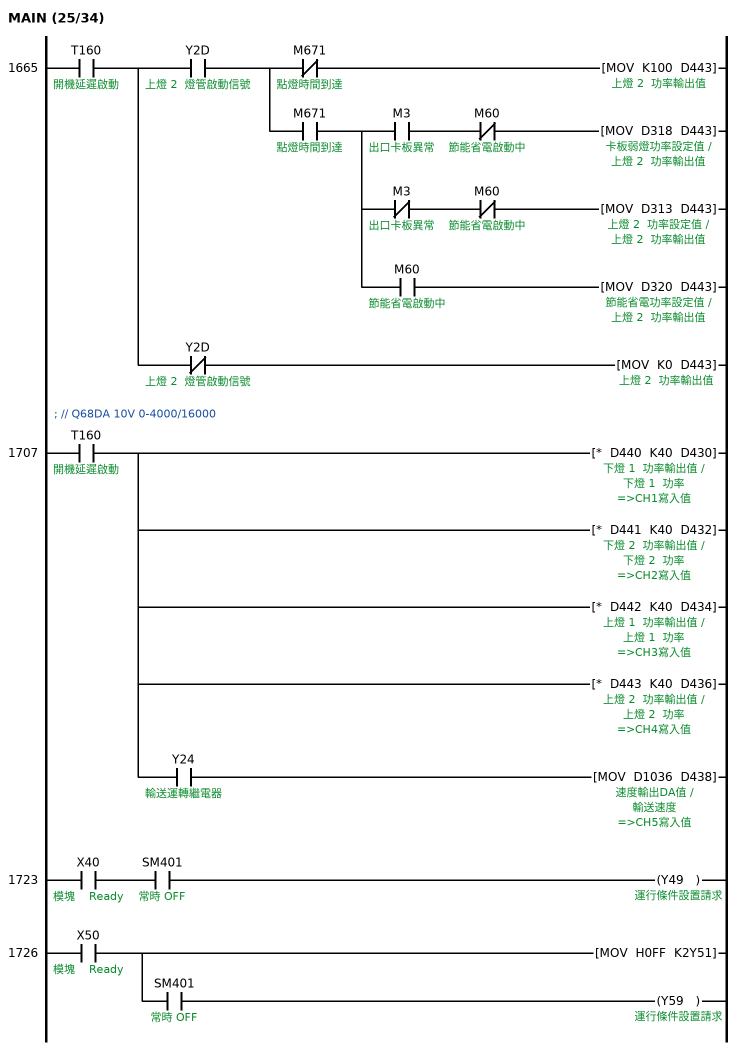
[picture p24: ladder of MAIN, rungs at steps 1665 to 1726]
1665  LD      T160  ; 開機延遲啟動
      MPS
      AND     Y2D  ; 上燈 2  燈管啟動信號
      MPS
      ANI     M671  ; 點燈時間到達
      MOV     K100 D443  ; 上燈 2  功率輸出值
      MPP
      AND     M671  ; 點燈時間到達
      MPS
      AND     M3  ; 出口卡板異常
      ANI     M60  ; 節能省電啟動中
      MOV     D318 D443
      MRD
      ANI     M3  ; 出口卡板異常
      ANI     M60  ; 節能省電啟動中
      MOV     D313 D443
      MPP
      AND     M60  ; 節能省電啟動中
      MOV     D320 D443
      MPP
      ANI     Y2D  ; 上燈 2  燈管啟動信號
      MOV     K0 D443
; // Q68DA 10V 0-4000/16000
1707  LD      T160  ; 開機延遲啟動
      *       D440 K40 D430  ; 下燈 1  功率  =>CH1寫入值
      *       D441 K40 D432  ; 下燈 2  功率  =>CH2寫入值
      *       D442 K40 D434  ; 上燈 1  功率  =>CH3寫入值
      *       D443 K40 D436  ; 上燈 2  功率  =>CH4寫入值
      AND     Y24  ; 輸送運轉繼電器
      MOV     D1036 D438  ; 速度輸出DA值 / 輸送速度      =>CH5寫入值
1723  LD      X40  ; 模塊    Ready
      AND     SM401  ; 常時 OFF
      OUT     Y49  ; 運行條件設置請求
1726  LD      X50  ; 模塊    Ready
      MOV     H0FF K2Y51  ; CH1輸出 允許/禁止標誌
      AND     SM401  ; 常時 OFF
      OUT     Y59  ; 運行條件設置請求
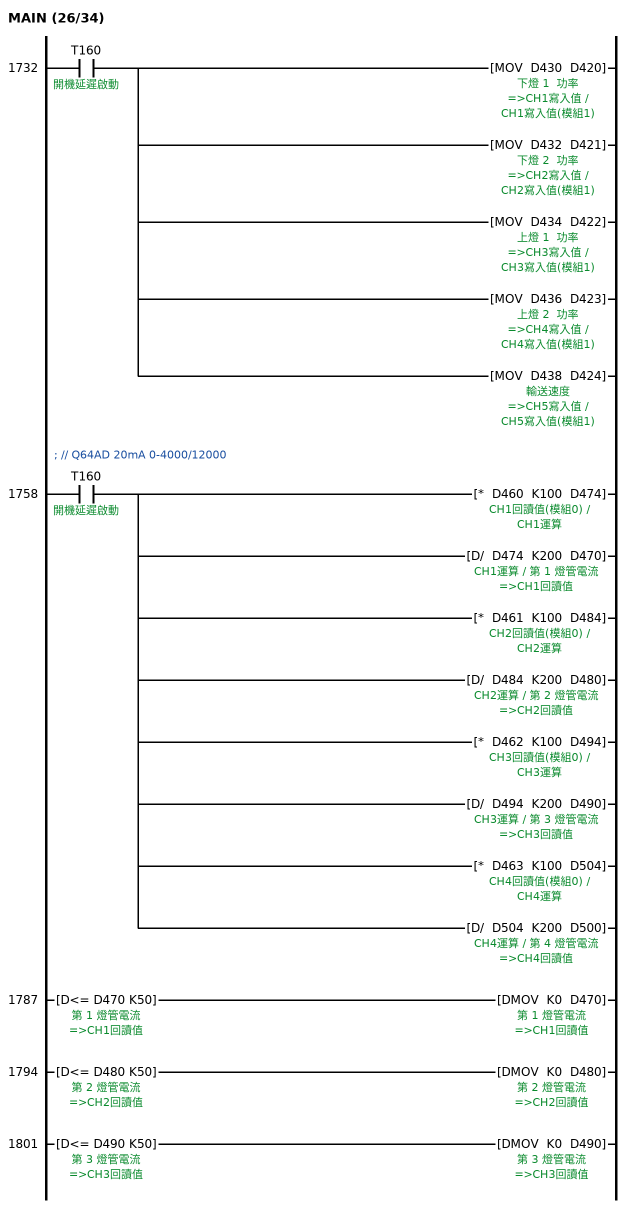
1732  LD      T160  ; 開機延遲啟動
      MOV     D430 D420  ; CH1寫入值(模組1)
      MOV     D432 D421  ; CH2寫入值(模組1)
      MOV     D434 D422  ; CH3寫入值(模組1)
      MOV     D436 D423  ; CH4寫入值(模組1)
      MOV     D438 D424  ; CH5寫入值(模組1)
; // Q64AD 20mA 0-4000/12000
1758  LD      T160  ; 開機延遲啟動
      *       D460 K100 D474  ; CH1回讀值(模組0) / CH1運算
      D/      D474 K200 D470  ; 第 1 燈管電流  =>CH1回讀值
      *       D461 K100 D484  ; CH2回讀值(模組0) / CH2運算
      D/      D484 K200 D480  ; 第 2 燈管電流  =>CH2回讀值
      *       D462 K100 D494  ; CH3回讀值(模組0) / CH3運算
      D/      D494 K200 D490  ; 第 3 燈管電流  =>CH3回讀值
      *       D463 K100 D504  ; CH4回讀值(模組0) / CH4運算
      D/      D504 K200 D500  ; 第 4 燈管電流  =>CH4回讀值
1787  LDD<=   D470 K50  ; 第 1 燈管電流  =>CH1回讀值
      DMOV    K0 D470
1794  LDD<=   D480 K50  ; 第 2 燈管電流  =>CH2回讀值
      DMOV    K0 D480
1801  LDD<=   D490 K50  ; 第 3 燈管電流  =>CH3回讀值
      DMOV    K0 D490
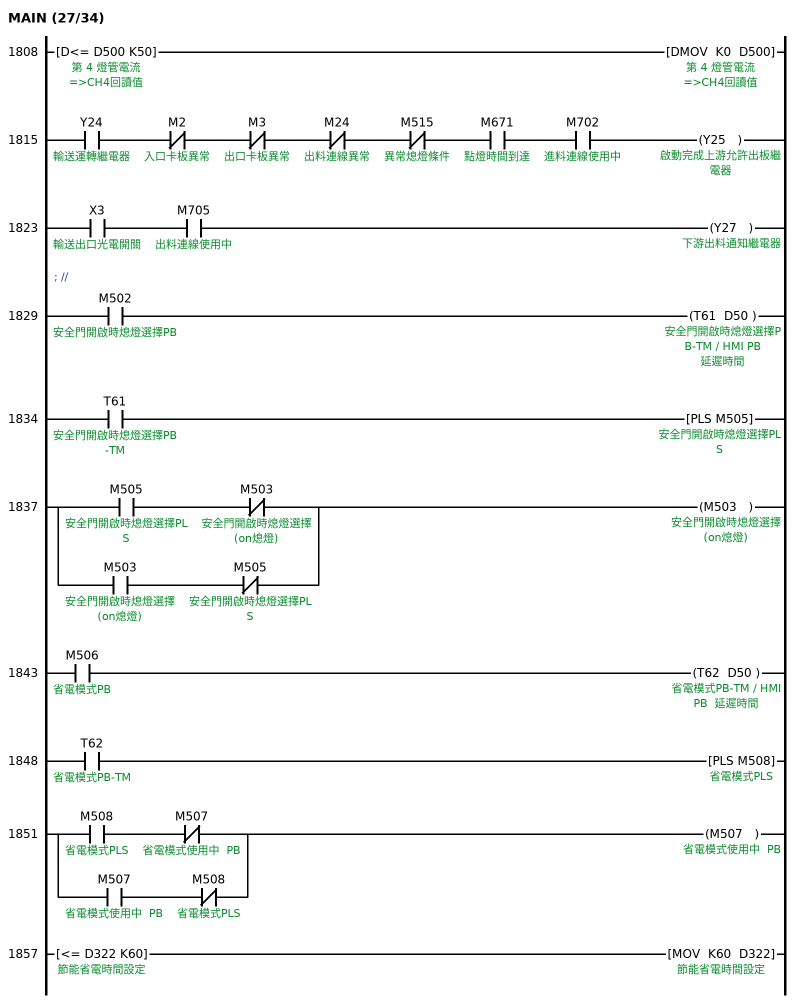
1808  LDD<=   D500 K50  ; 第 4 燈管電流  =>CH4回讀值
      DMOV    K0 D500
1815  LD      Y24  ; 輸送運轉繼電器
      ANI     M2  ; 入口卡板異常
      ANI     M3  ; 出口卡板異常
      ANI     M24  ; 出料連線異常
      ANI     M515  ; 異常熄燈條件
      AND     M671  ; 點燈時間到達
      AND     M702  ; 進料連線使用中
      OUT     Y25  ; 啟動完成上游允許出板繼電器
1823  LD      X3  ; 輸送出口光電開關
      AND     M705  ; 出料連線使用中
      OUT     Y27  ; 下游出料通知繼電器
; //
1829  LD      M502  ; 安全門開啟時熄燈選擇PB
      OUT     T61 D50  ; 安全門開啟時熄燈選擇PB-TM / HMI PB  延遲時間
1834  LD      T61  ; 安全門開啟時熄燈選擇PB-TM
      PLS     M505  ; 安全門開啟時熄燈選擇PLS
1837  LD      M505  ; 安全門開啟時熄燈選擇PLS
      ANI     M503  ; 安全門開啟時熄燈選擇    (on熄燈)
      LD      M503  ; 安全門開啟時熄燈選擇    (on熄燈)
      ANI     M505  ; 安全門開啟時熄燈選擇PLS
      ORB
      OUT     M503  ; 安全門開啟時熄燈選擇    (on熄燈)
1843  LD      M506  ; 省電模式PB
      OUT     T62 D50  ; 省電模式PB-TM / HMI PB  延遲時間
1848  LD      T62  ; 省電模式PB-TM
      PLS     M508  ; 省電模式PLS
1851  LD      M508  ; 省電模式PLS
      ANI     M507  ; 省電模式使用中  PB
      LD      M507  ; 省電模式使用中  PB
      ANI     M508  ; 省電模式PLS
      ORB
      OUT     M507  ; 省電模式使用中  PB
1857  LD<=    D322 K60  ; 節能省電時間設定
      MOV     K60 D322
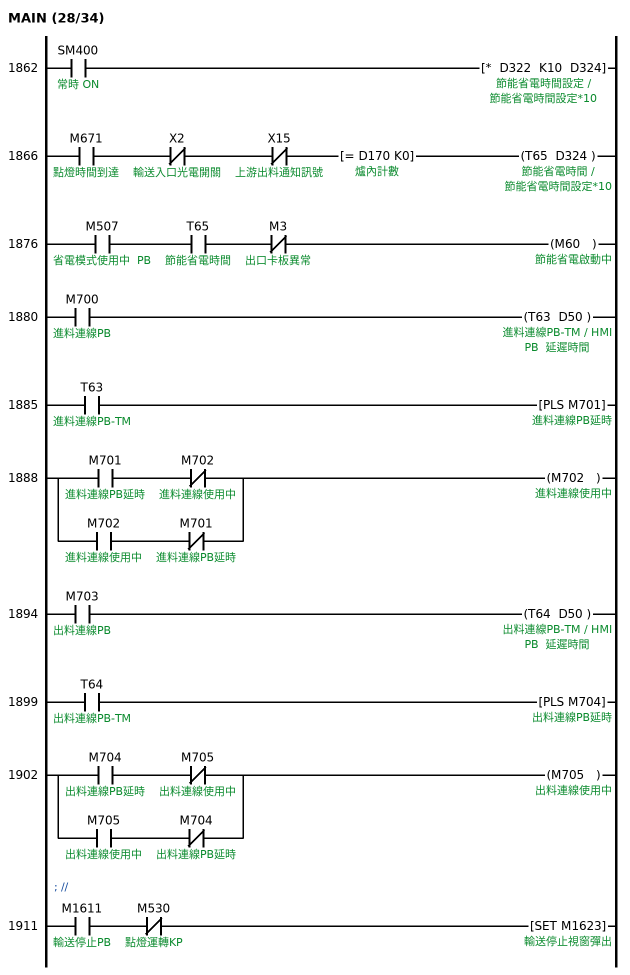
1862  LD      SM400  ; 常時 ON
      *       D322 K10 D324  ; 節能省電時間設定*10
1866  LD      M671  ; 點燈時間到達
      ANI     X2  ; 輸送入口光電開關
      ANI     X15  ; 上游出料通知訊號
      AND=    D170 K0  ; 爐內計數
      OUT     T65 D324  ; 節能省電時間 / 節能省電時間設定*10
1876  LD      M507  ; 省電模式使用中  PB
      AND     T65  ; 節能省電時間
      ANI     M3  ; 出口卡板異常
      OUT     M60  ; 節能省電啟動中
1880  LD      M700  ; 進料連線PB
      OUT     T63 D50  ; 進料連線PB-TM / HMI PB  延遲時間
1885  LD      T63  ; 進料連線PB-TM
      PLS     M701  ; 進料連線PB延時
1888  LD      M701  ; 進料連線PB延時
      ANI     M702  ; 進料連線使用中
      LD      M702  ; 進料連線使用中
      ANI     M701  ; 進料連線PB延時
      ORB
      OUT     M702  ; 進料連線使用中
1894  LD      M703  ; 出料連線PB
      OUT     T64 D50  ; 出料連線PB-TM / HMI PB  延遲時間
1899  LD      T64  ; 出料連線PB-TM
      PLS     M704  ; 出料連線PB延時
1902  LD      M704  ; 出料連線PB延時
      ANI     M705  ; 出料連線使用中
      LD      M705  ; 出料連線使用中
      ANI     M704  ; 出料連線PB延時
      ORB
      OUT     M705  ; 出料連線使用中
; //
1911  LD      M1611  ; 輸送停止PB
      ANI     M530  ; 點燈運轉KP
      SET     M1623  ; 輸送停止視窗彈出
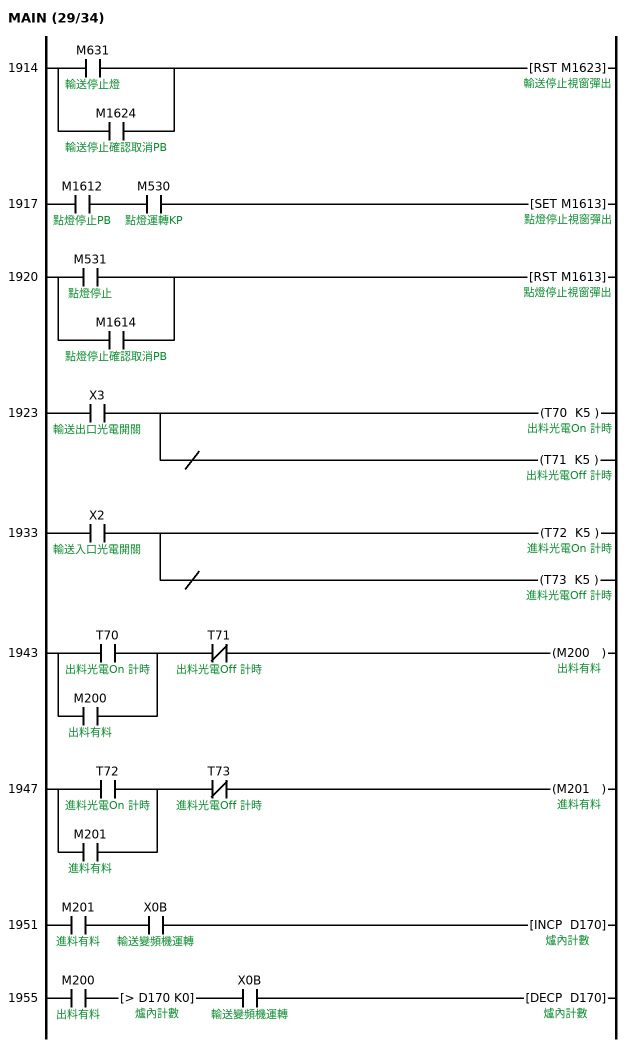
1914  LD      M631  ; 輸送停止燈
      OR      M1624  ; 輸送停止確認取消PB
      RST     M1623  ; 輸送停止視窗彈出
1917  LD      M1612  ; 點燈停止PB
      AND     M530  ; 點燈運轉KP
      SET     M1613  ; 點燈停止視窗彈出
1920  LD      M531  ; 點燈停止
      OR      M1614  ; 點燈停止確認取消PB
      RST     M1613  ; 點燈停止視窗彈出
1923  LD      X3  ; 輸送出口光電開關
      OUT     T70 K5  ; 出料光電On 計時
      INV
      OUT     T71 K5  ; 出料光電Off 計時
1933  LD      X2  ; 輸送入口光電開關
      OUT     T72 K5  ; 進料光電On 計時
      INV
      OUT     T73 K5  ; 進料光電Off 計時
1943  LD      T70  ; 出料光電On 計時
      OR      M200  ; 出料有料
      ANI     T71  ; 出料光電Off 計時
      OUT     M200  ; 出料有料
1947  LD      T72  ; 進料光電On 計時
      OR      M201  ; 進料有料
      ANI     T73  ; 進料光電Off 計時
      OUT     M201  ; 進料有料
1951  LD      M201  ; 進料有料
      AND     X0B  ; 輸送變頻機運轉
      INCP    D170
1955  LD      M200  ; 出料有料
      AND>    D170 K0  ; 爐內計數
      AND     X0B  ; 輸送變頻機運轉
      DECP    D170
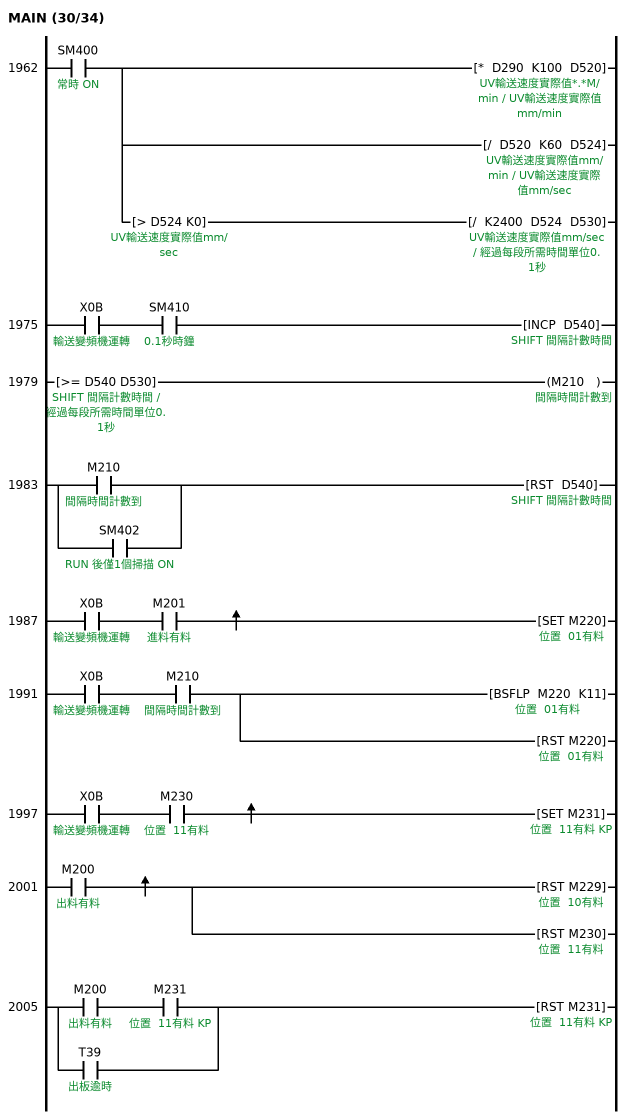
1962  LD      SM400  ; 常時 ON
      *       D290 K100 D520  ; UV輸送速度實際值mm/min
      /       D520 K60 D524  ; UV輸送速度實際值mm/sec
      AND>    D524 K0  ; UV輸送速度實際值mm/sec
      /       K2400 D524 D530  ; 經過每段所需時間單位0.1秒
1975  LD      X0B  ; 輸送變頻機運轉
      AND     SM410  ; 0.1秒時鐘
      INCP    D540  ; SHIFT 間隔計數時間
1979  LD>=    D540 D530  ; SHIFT 間隔計數時間 / 經過每段所需時間單位0.1秒
      OUT     M210  ; 間隔時間計數到
1983  LD      M210  ; 間隔時間計數到
      OR      SM402  ; RUN 後僅1個掃描 ON
      RST     D540  ; SHIFT 間隔計數時間
1987  LD      X0B  ; 輸送變頻機運轉
      AND     M201  ; 進料有料
      MEP
      SET     M220  ; 位置  01有料
1991  LD      X0B  ; 輸送變頻機運轉
      AND     M210  ; 間隔時間計數到
      BSFLP   M220 K11
      RST     M220  ; 位置  01有料
1997  LD      X0B  ; 輸送變頻機運轉
      AND     M230  ; 位置  11有料
      MEP
      SET     M231  ; 位置  11有料 KP
2001  LD      M200  ; 出料有料
      MEP
      RST     M229  ; 位置  10有料
      RST     M230  ; 位置  11有料
2005  LD      M200  ; 出料有料
      AND     M231  ; 位置  11有料 KP
      OR      T39  ; 出板逾時
      RST     M231  ; 位置  11有料 KP
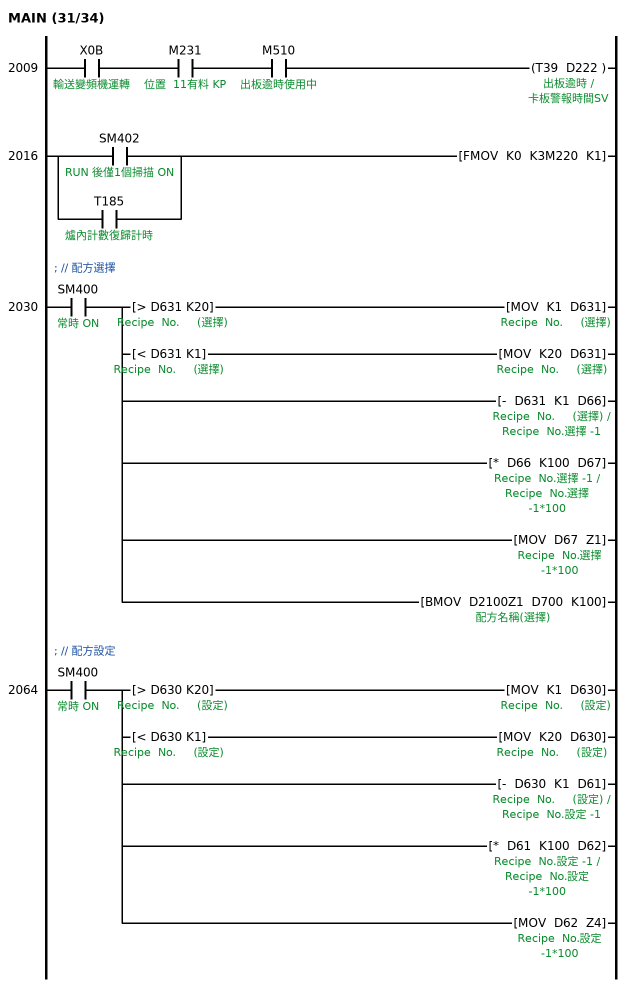
2009  LD      X0B  ; 輸送變頻機運轉
      AND     M231  ; 位置  11有料 KP
      AND     M510  ; 出板逾時使用中
      OUT     T39 D222  ; 出板逾時 / 卡板警報時間SV
2016  LD      SM402  ; RUN 後僅1個掃描 ON
      OR      T185  ; 爐內計數復歸計時
      FMOV    K0 K3M220 K1
; // 配方選擇
2030  LD      SM400  ; 常時 ON
      MPS
      AND>    D631 K20  ; Recipe  No.     (選擇)
      MOV     K1 D631
      MRD
      AND<    D631 K1  ; Recipe  No.     (選擇)
      MOV     K20 D631
      MPP
      -       D631 K1 D66  ; Recipe  No.選擇 -1
      *       D66 K100 D67  ; Recipe  No.選擇 -1*100
      MOV     D67 Z1
      BMOV    D2100Z1 D700 K100  ; 配方名稱(選擇)
; // 配方設定
2064  LD      SM400  ; 常時 ON
      MPS
      AND>    D630 K20  ; Recipe  No.     (設定)
      MOV     K1 D630
      MRD
      AND<    D630 K1  ; Recipe  No.     (設定)
      MOV     K20 D630
      MPP
      -       D630 K1 D61  ; Recipe  No.設定 -1
      *       D61 K100 D62  ; Recipe  No.設定 -1*100
      MOV     D62 Z4
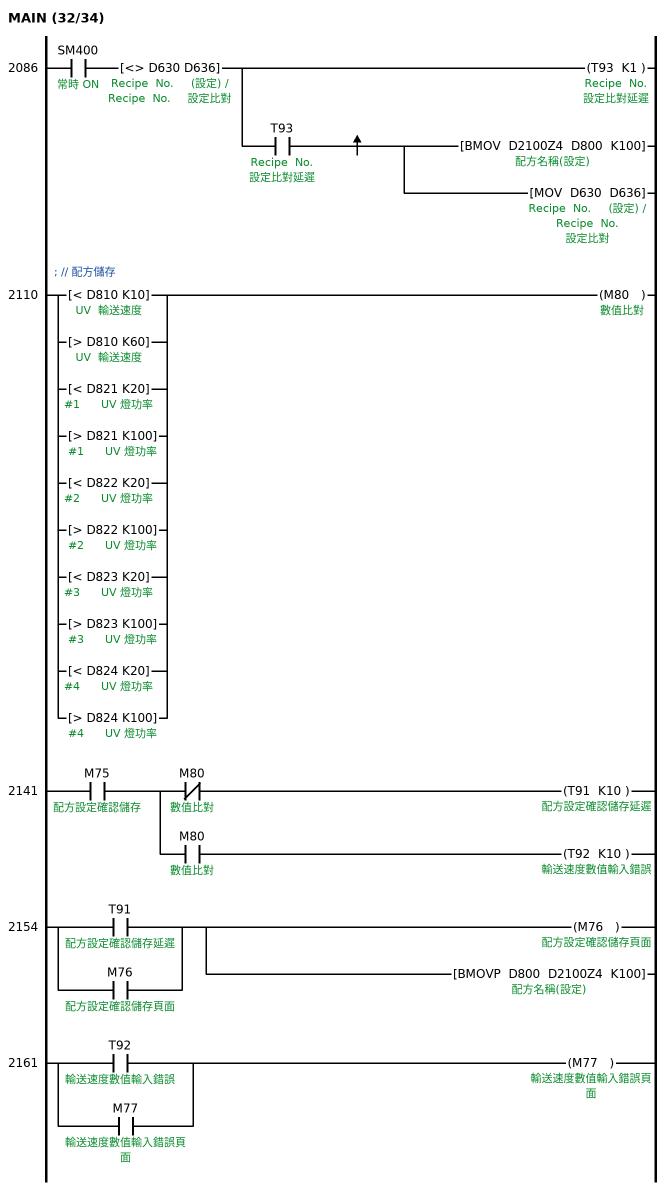
2086  LD      SM400  ; 常時 ON
      AND<>   D630 D636  ; Recipe  No.     (設定) / Recipe  No.     設定比對
      OUT     T93 K1  ; Recipe  No.     設定比對延遲
      AND     T93  ; Recipe  No.     設定比對延遲
      MEP
      BMOV    D2100Z4 D800 K100  ; 配方名稱(設定)
      MOV     D630 D636
; // 配方儲存
2110  LD<     D810 K10  ; UV  輸送速度
      OR>     D810 K60  ; UV  輸送速度
      OR<     D821 K20  ; #1      UV 燈功率
      OR>     D821 K100  ; #1      UV 燈功率
      OR<     D822 K20  ; #2      UV 燈功率
      OR>     D822 K100  ; #2      UV 燈功率
      OR<     D823 K20  ; #3      UV 燈功率
      OR>     D823 K100  ; #3      UV 燈功率
      OR<     D824 K20  ; #4      UV 燈功率
      OR>     D824 K100  ; #4      UV 燈功率
      OUT     M80  ; 數值比對
2141  LD      M75  ; 配方設定確認儲存
      MPS
      ANI     M80  ; 數值比對
      OUT     T91 K10  ; 配方設定確認儲存延遲
      MPP
      AND     M80  ; 數值比對
      OUT     T92 K10  ; 輸送速度數值輸入錯誤
2154  LD      T91  ; 配方設定確認儲存延遲
      OR      M76  ; 配方設定確認儲存頁面
      OUT     M76  ; 配方設定確認儲存頁面
      BMOVP   D800 D2100Z4 K100
2161  LD      T92  ; 輸送速度數值輸入錯誤
      OR      M77  ; 輸送速度數值輸入錯誤頁面
      OUT     M77  ; 輸送速度數值輸入錯誤頁面
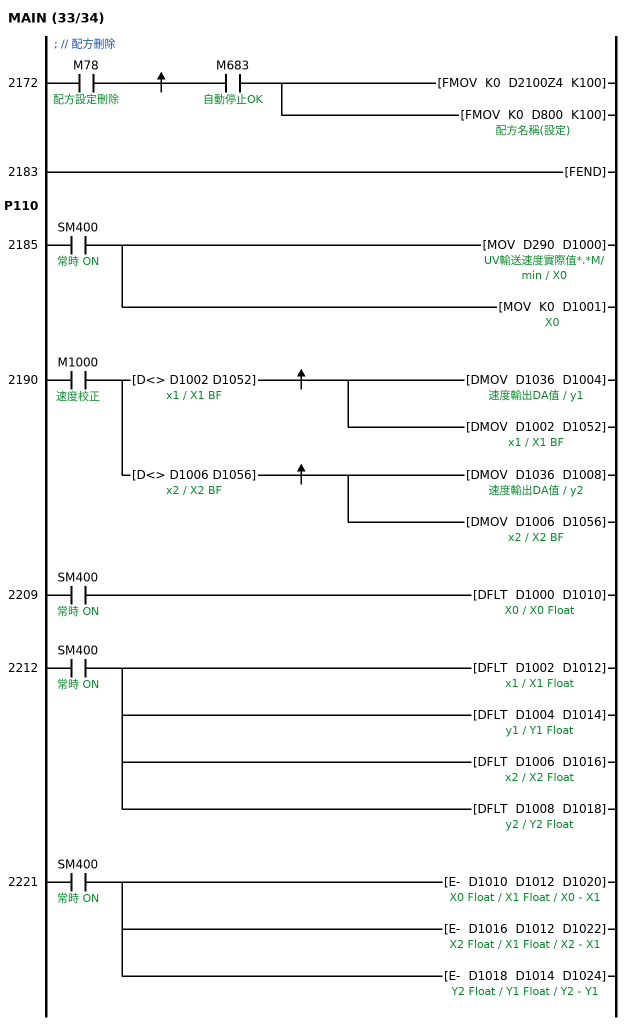
; // 配方刪除
2172  LD      M78  ; 配方設定刪除
      MEP
      AND     M683  ; 自動停止OK
      FMOV    K0 D2100Z4 K100
      FMOV    K0 D800 K100
2183  FEND
      P110
2185  LD      SM400  ; 常時 ON
      MOV     D290 D1000  ; X0
      MOV     K0 D1001  ; X0
2190  LD      M1000  ; 速度校正
      MPS
      ANDD<>  D1002 D1052  ; x1 / X1 BF
      MEP
      DMOV    D1036 D1004  ; y1
      DMOV    D1002 D1052
      MPP
      ANDD<>  D1006 D1056  ; x2 / X2 BF
      MEP
      DMOV    D1036 D1008  ; y2
      DMOV    D1006 D1056
2209  LD      SM400  ; 常時 ON
      DFLT    D1000 D1010  ; X0 Float
2212  LD      SM400  ; 常時 ON
      DFLT    D1002 D1012  ; X1 Float
      DFLT    D1004 D1014  ; Y1 Float
      DFLT    D1006 D1016  ; X2 Float
      DFLT    D1008 D1018  ; Y2 Float
2221  LD      SM400  ; 常時 ON
      E-      D1010 D1012 D1020  ; X0 - X1
      E-      D1016 D1012 D1022  ; X2 - X1
      E-      D1018 D1014 D1024  ; Y2 - Y1
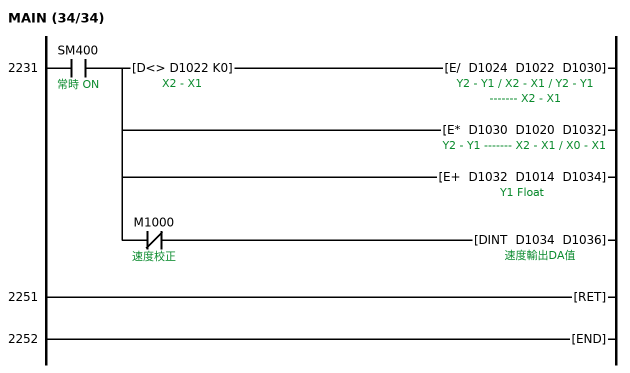
2231  LD      SM400  ; 常時 ON
      MPS
      ANDD<>  D1022 K0  ; X2 - X1
      E/      D1024 D1022 D1030  ; Y2 - Y1 ------- X2 - X1
      MPP
      E*      D1030 D1020 D1032
      E+      D1032 D1014 D1034
      ANI     M1000  ; 速度校正
      DINT    D1034 D1036
2251  RET
2252  END
END_PROGRAM

PROGRAM SECS
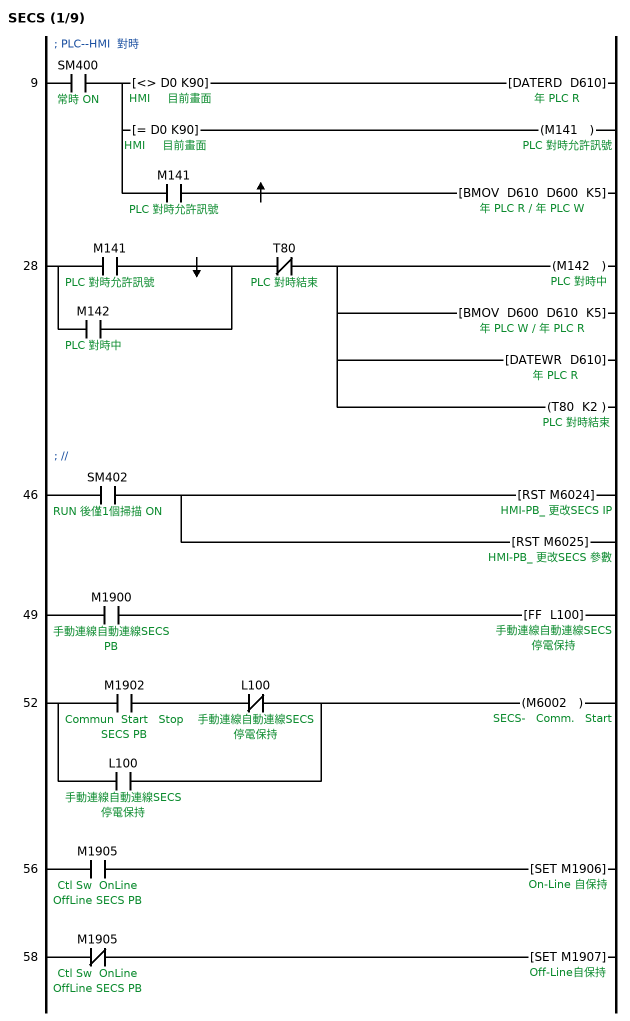
; PLC--HMI  對時
9     LD      SM400  ; 常時 ON
      MPS
      AND<>   D0 K90  ; HMI     目前畫面
      DATERD  D610  ; 年 PLC R
      MRD
      AND=    D0 K90  ; HMI     目前畫面
      OUT     M141  ; PLC 對時允許訊號
      MPP
      AND     M141  ; PLC 對時允許訊號
      MEP
      BMOV    D610 D600 K5  ; 年 PLC W
28    LD      M141  ; PLC 對時允許訊號
      MEF
      OR      M142  ; PLC 對時中
      ANI     T80  ; PLC 對時結束
      OUT     M142  ; PLC 對時中
      BMOV    D600 D610 K5
      DATEWR  D610
      OUT     T80 K2  ; PLC 對時結束
; //
46    LD      SM402  ; RUN 後僅1個掃描 ON
      RST     M6024  ; HMI-PB_ 更改SECS IP
      RST     M6025  ; HMI-PB_ 更改SECS 參數
49    LD      M1900  ; 手動連線自動連線SECS PB
      FF      L100  ; 手動連線自動連線SECS    停電保持
52    LD      M1902  ; Commun  Start   Stop    SECS PB
      ANI     L100  ; 手動連線自動連線SECS    停電保持
      OR      L100  ; 手動連線自動連線SECS    停電保持
      OUT     M6002  ; SECS-   Comm.   Start
56    LD      M1905  ; Ctl Sw  OnLine  OffLine SECS PB
      SET     M1906  ; On-Line 自保持
58    LDI     M1905  ; Ctl Sw  OnLine  OffLine SECS PB
      SET     M1907  ; Off-Line自保持
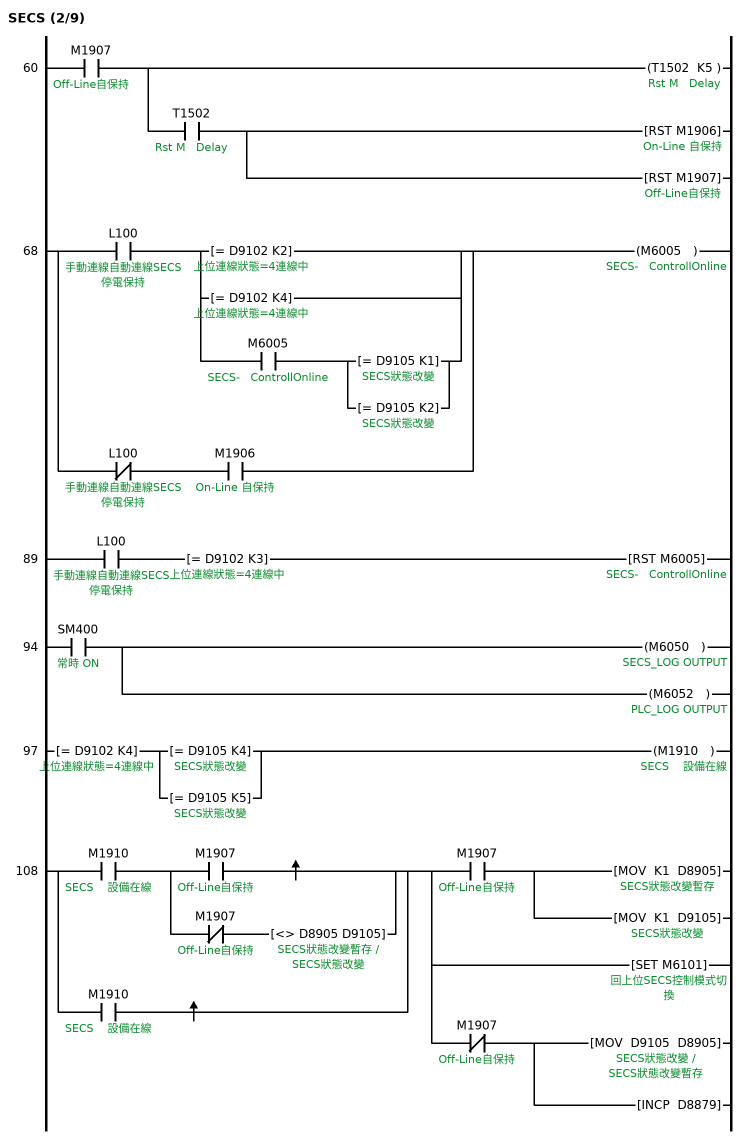
60    LD      M1907  ; Off-Line自保持
      OUT     T1502 K5  ; Rst M   Delay
      AND     T1502  ; Rst M   Delay
      RST     M1906  ; On-Line 自保持
      RST     M1907  ; Off-Line自保持
68    LD      L100  ; 手動連線自動連線SECS    停電保持
      LD=     D9102 K2  ; 上位連線狀態=4連線中
      OR=     D9102 K4  ; 上位連線狀態=4連線中
      LD      M6005  ; SECS-   ControllOnline
      LD=     D9105 K1  ; SECS狀態改變
      OR=     D9105 K2  ; SECS狀態改變
      ANB
      ORB
      ANB
      LDI     L100  ; 手動連線自動連線SECS    停電保持
      AND     M1906  ; On-Line 自保持
      ORB
      OUT     M6005  ; SECS-   ControllOnline
89    LD      L100  ; 手動連線自動連線SECS    停電保持
      AND=    D9102 K3  ; 上位連線狀態=4連線中
      RST     M6005  ; SECS-   ControllOnline
94    LD      SM400  ; 常時 ON
      OUT     M6050  ; SECS_LOG OUTPUT
      OUT     M6052  ; PLC_LOG OUTPUT
97    LD=     D9102 K4  ; 上位連線狀態=4連線中
      LD=     D9105 K4  ; SECS狀態改變
      OR=     D9105 K5  ; SECS狀態改變
      ANB
      OUT     M1910  ; SECS    設備在線
108   LD      M1910  ; SECS    設備在線
      LD      M1907  ; Off-Line自保持
      MEP
      LDI     M1907  ; Off-Line自保持
      AND<>   D8905 D9105  ; SECS狀態改變暫存 / SECS狀態改變
      ORB
      ANB
      LD      M1910  ; SECS    設備在線
      MEP
      ORB
      MPS
      AND     M1907  ; Off-Line自保持
      MOV     K1 D8905
      MOV     K1 D9105
      MPP
      SET     M6101  ; 回上位SECS控制模式切換
      ANI     M1907  ; Off-Line自保持
      MOV     D9105 D8905
      INCP    D8879
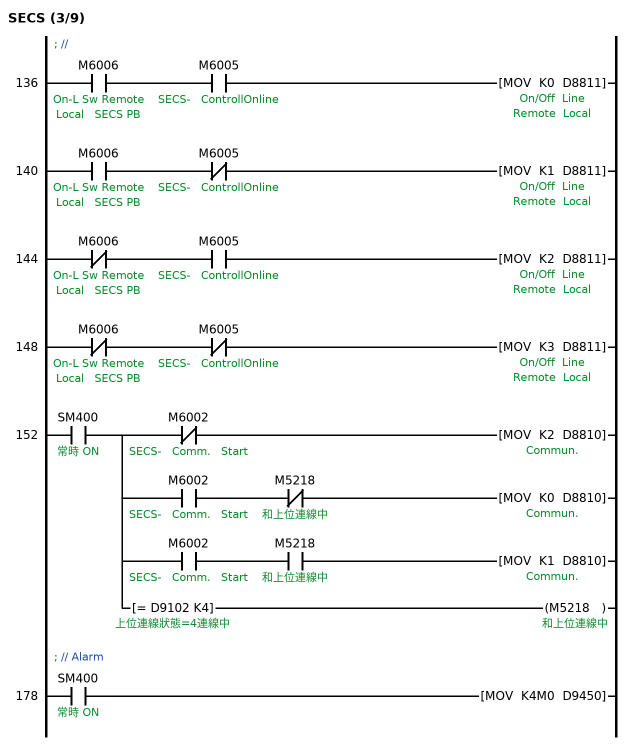
; //
136   LD      M6006  ; On-L Sw Remote  Local   SECS PB
      AND     M6005  ; SECS-   ControllOnline
      MOV     K0 D8811  ; On/Off  Line    Remote  Local
140   LD      M6006  ; On-L Sw Remote  Local   SECS PB
      ANI     M6005  ; SECS-   ControllOnline
      MOV     K1 D8811
144   LDI     M6006  ; On-L Sw Remote  Local   SECS PB
      AND     M6005  ; SECS-   ControllOnline
      MOV     K2 D8811
148   LDI     M6006  ; On-L Sw Remote  Local   SECS PB
      ANI     M6005  ; SECS-   ControllOnline
      MOV     K3 D8811
152   LD      SM400  ; 常時 ON
      MPS
      ANI     M6002  ; SECS-   Comm.   Start
      MOV     K2 D8810  ; Commun.
      MRD
      AND     M6002  ; SECS-   Comm.   Start
      ANI     M5218  ; 和上位連線中
      MOV     K0 D8810
      MRD
      AND     M6002  ; SECS-   Comm.   Start
      AND     M5218  ; 和上位連線中
      MOV     K1 D8810
      MPP
      AND=    D9102 K4  ; 上位連線狀態=4連線中
      OUT     M5218  ; 和上位連線中
; // Alarm
178   LD      SM400  ; 常時 ON
      MOV     K4M0 D9450  ; 緊急停止開關異常
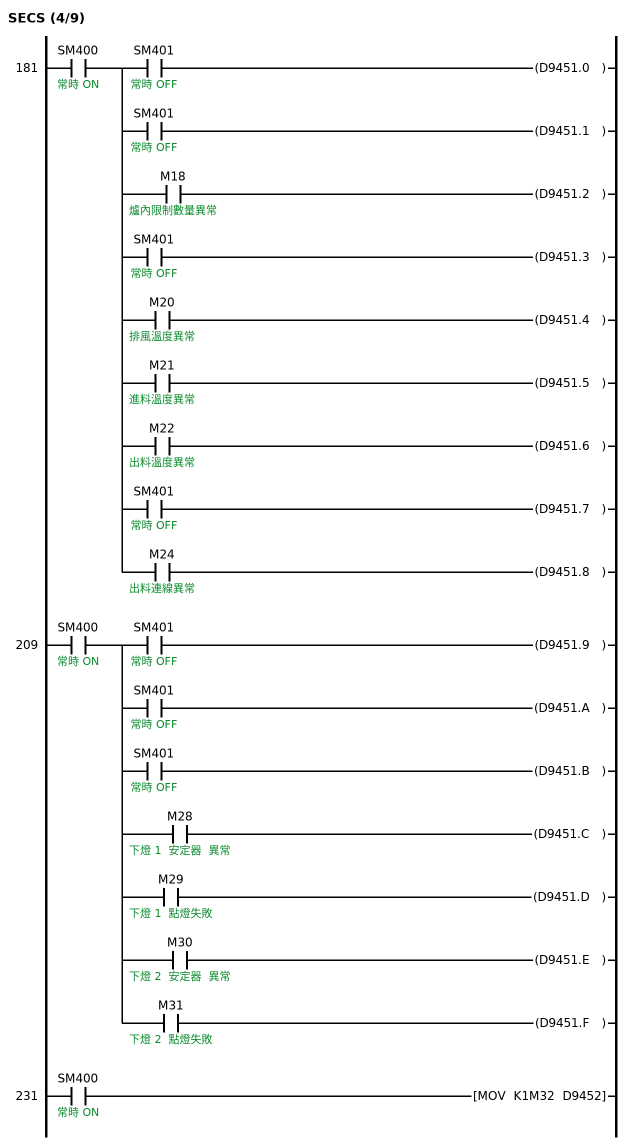
181   LD      SM400  ; 常時 ON
      MPS
      AND     SM401  ; 常時 OFF
      OUT     D9451.0
      MRD
      AND     SM401  ; 常時 OFF
      OUT     D9451.1
      MRD
      AND     M18  ; 爐內限制數量異常
      OUT     D9451.2
      MRD
      AND     SM401  ; 常時 OFF
      OUT     D9451.3
      MRD
      AND     M20  ; 排風溫度異常
      OUT     D9451.4
      MRD
      AND     M21  ; 進料溫度異常
      OUT     D9451.5
      MRD
      AND     M22  ; 出料溫度異常
      OUT     D9451.6
      MRD
      AND     SM401  ; 常時 OFF
      OUT     D9451.7
      MPP
      AND     M24  ; 出料連線異常
      OUT     D9451.8
209   LD      SM400  ; 常時 ON
      MPS
      AND     SM401  ; 常時 OFF
      OUT     D9451.9
      MRD
      AND     SM401  ; 常時 OFF
      OUT     D9451.A
      MRD
      AND     SM401  ; 常時 OFF
      OUT     D9451.B
      MRD
      AND     M28  ; 下燈 1  安定器  異常
      OUT     D9451.C
      MRD
      AND     M29  ; 下燈 1  點燈失敗
      OUT     D9451.D
      MRD
      AND     M30  ; 下燈 2  安定器  異常
      OUT     D9451.E
      MPP
      AND     M31  ; 下燈 2  點燈失敗
      OUT     D9451.F
231   LD      SM400  ; 常時 ON
      MOV     K1M32 D9452  ; 上燈 1  安定器  異常
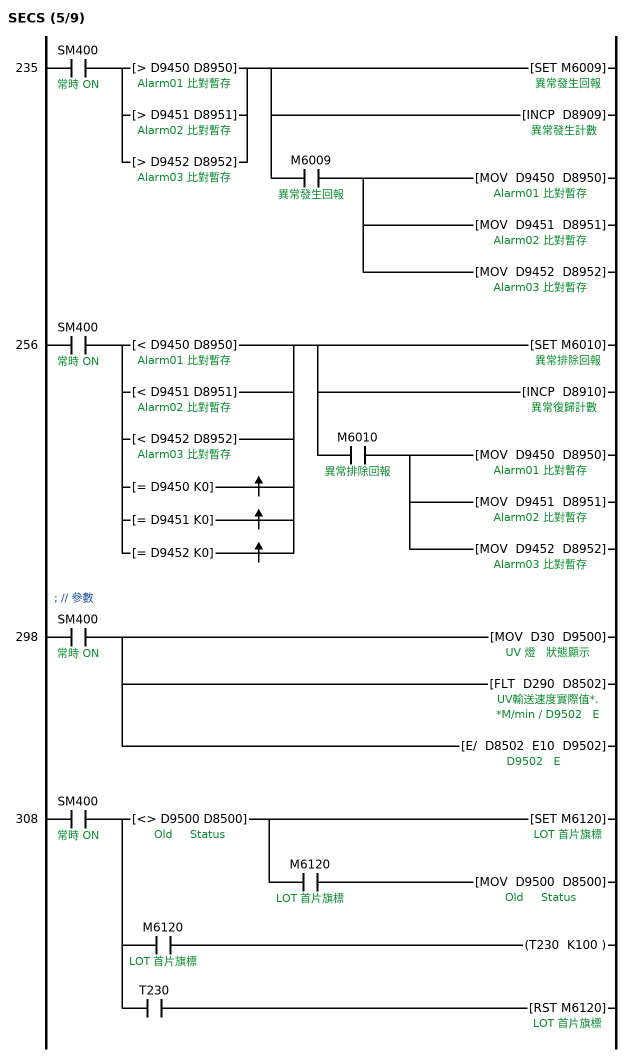
235   LD      SM400  ; 常時 ON
      LD>     D9450 D8950  ; Alarm01 比對暫存
      OR>     D9451 D8951  ; Alarm02 比對暫存
      OR>     D9452 D8952  ; Alarm03 比對暫存
      ANB
      SET     M6009  ; 異常發生回報
      INCP    D8909  ; 異常發生計數
      AND     M6009  ; 異常發生回報
      MOV     D9450 D8950
      MOV     D9451 D8951
      MOV     D9452 D8952
256   LD      SM400  ; 常時 ON
      LD<     D9450 D8950  ; Alarm01 比對暫存
      OR<     D9451 D8951  ; Alarm02 比對暫存
      OR<     D9452 D8952  ; Alarm03 比對暫存
      LD=     D9450 K0
      MEP
      ORB
      LD=     D9451 K0
      MEP
      ORB
      LD=     D9452 K0
      MEP
      ORB
      ANB
      SET     M6010  ; 異常排除回報
      INCP    D8910  ; 異常復歸計數
      AND     M6010  ; 異常排除回報
      MOV     D9450 D8950
      MOV     D9451 D8951
      MOV     D9452 D8952
; // 參數
298   LD      SM400  ; 常時 ON
      MOV     D30 D9500  ; UV 燈   狀態顯示
      FLT     D290 D8502  ; UV輸送速度實際值*.*M/min / D9502   E
      E/      D8502 E10 D9502
308   LD      SM400  ; 常時 ON
      MPS
      AND<>   D9500 D8500  ; Old     Status
      SET     M6120  ; LOT 首片旗標
      AND     M6120  ; LOT 首片旗標
      MOV     D9500 D8500
      MRD
      AND     M6120  ; LOT 首片旗標
      OUT     T230 K100
      MPP
      AND     T230
      RST     M6120  ; LOT 首片旗標
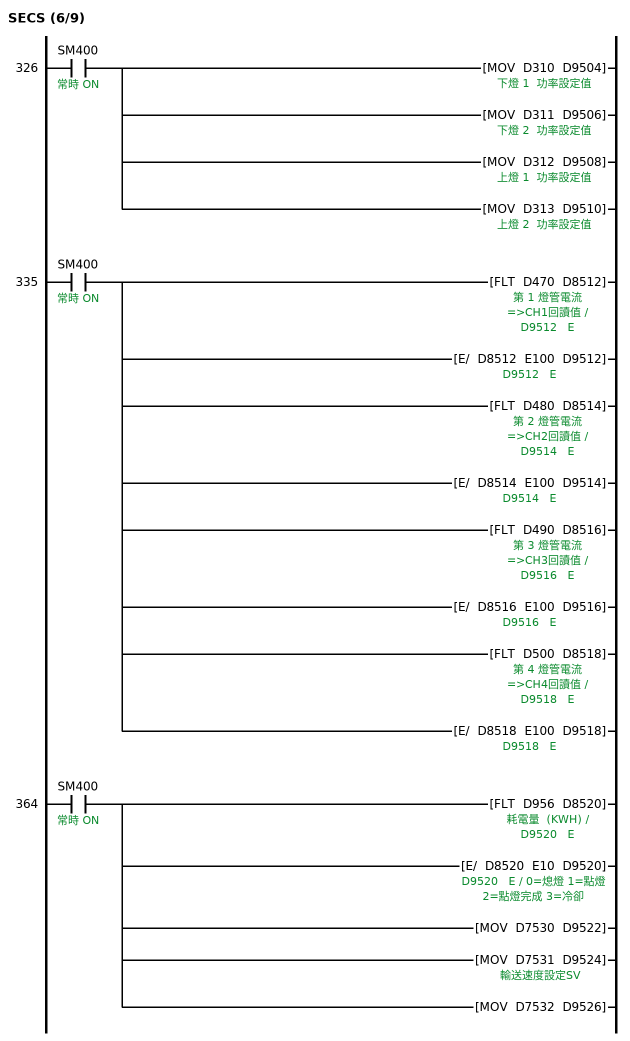
326   LD      SM400  ; 常時 ON
      MOV     D310 D9504  ; 下燈 1  功率設定值
      MOV     D311 D9506  ; 下燈 2  功率設定值
      MOV     D312 D9508  ; 上燈 1  功率設定值
      MOV     D313 D9510  ; 上燈 2  功率設定值
335   LD      SM400  ; 常時 ON
      FLT     D470 D8512  ; 第 1 燈管電流  =>CH1回讀值 / D9512   E
      E/      D8512 E100 D9512
      FLT     D480 D8514  ; 第 2 燈管電流  =>CH2回讀值 / D9514   E
      E/      D8514 E100 D9514
      FLT     D490 D8516  ; 第 3 燈管電流  =>CH3回讀值 / D9516   E
      E/      D8516 E100 D9516
      FLT     D500 D8518  ; 第 4 燈管電流  =>CH4回讀值 / D9518   E
      E/      D8518 E100 D9518
364   LD      SM400  ; 常時 ON
      FLT     D956 D8520  ; 耗電量  (KWH) / D9520   E
      E/      D8520 E10 D9520  ; 0=熄燈 1=點燈 2=點燈完成 3=冷卻
      MOV     D7530 D9522
      MOV     D7531 D9524  ; 輸送速度設定SV
      MOV     D7532 D9526
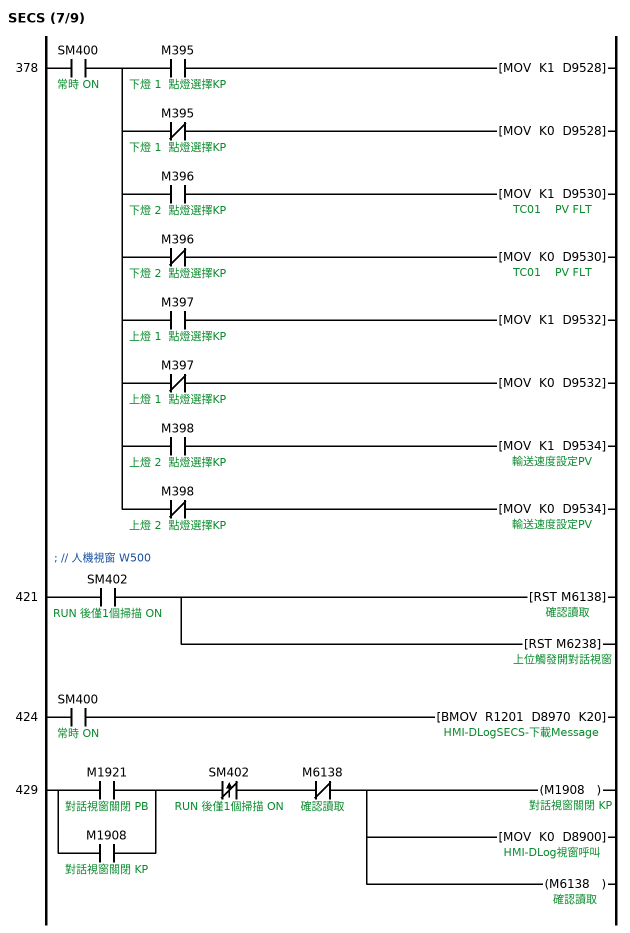
378   LD      SM400  ; 常時 ON
      MPS
      AND     M395  ; 下燈 1  點燈選擇KP
      MOV     K1 D9528
      MRD
      ANI     M395  ; 下燈 1  點燈選擇KP
      MOV     K0 D9528
      MRD
      AND     M396  ; 下燈 2  點燈選擇KP
      MOV     K1 D9530  ; TC01    PV FLT
      MRD
      ANI     M396  ; 下燈 2  點燈選擇KP
      MOV     K0 D9530
      MRD
      AND     M397  ; 上燈 1  點燈選擇KP
      MOV     K1 D9532
      MRD
      ANI     M397  ; 上燈 1  點燈選擇KP
      MOV     K0 D9532
      MRD
      AND     M398  ; 上燈 2  點燈選擇KP
      MOV     K1 D9534  ; 輸送速度設定PV
      MPP
      ANI     M398  ; 上燈 2  點燈選擇KP
      MOV     K0 D9534
; // 人機視窗 W500
421   LD      SM402  ; RUN 後僅1個掃描 ON
      RST     M6138  ; 確認讀取
      RST     M6238  ; 上位觸發開對話視窗
424   LD      SM400  ; 常時 ON
      BMOV    R1201 D8970 K20  ; HMI-DLogSECS-下載Message
429   LD      M1921  ; 對話視窗關閉 PB
      OR      M1908  ; 對話視窗關閉 KP
      ANDPI   SM402  ; RUN 後僅1個掃描 ON
      ANI     M6138  ; 確認讀取
      OUT     M1908  ; 對話視窗關閉 KP
      MOV     K0 D8900  ; HMI-DLog視窗呼叫
      OUT     M6138  ; 確認讀取
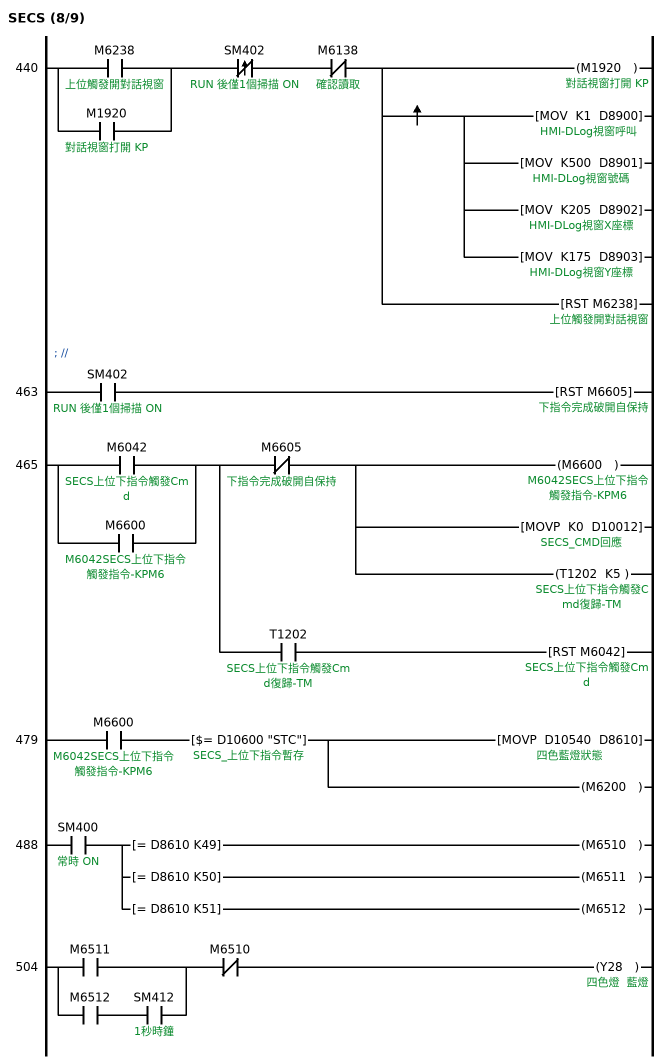
440   LD      M6238  ; 上位觸發開對話視窗
      OR      M1920  ; 對話視窗打開 KP
      ANDPI   SM402  ; RUN 後僅1個掃描 ON
      ANI     M6138  ; 確認讀取
      OUT     M1920  ; 對話視窗打開 KP
      MPS
      MEP
      MOV     K1 D8900
      MOV     K500 D8901  ; HMI-DLog視窗號碼
      MOV     K205 D8902  ; HMI-DLog視窗X座標
      MOV     K175 D8903  ; HMI-DLog視窗Y座標
      MPP
      RST     M6238  ; 上位觸發開對話視窗
; //
463   LD      SM402  ; RUN 後僅1個掃描 ON
      RST     M6605  ; 下指令完成破開自保持
465   LD      M6042  ; SECS上位下指令觸發Cmd
      OR      M6600  ; M6042SECS上位下指令觸發指令-KPM6
      MPS
      ANI     M6605  ; 下指令完成破開自保持
      OUT     M6600  ; M6042SECS上位下指令觸發指令-KPM6
      MOVP    K0 D10012  ; SECS_CMD回應
      OUT     T1202 K5  ; SECS上位下指令觸發Cmd復歸-TM
      MPP
      AND     T1202  ; SECS上位下指令觸發Cmd復歸-TM
      RST     M6042  ; SECS上位下指令觸發Cmd
479   LD      M6600  ; M6042SECS上位下指令觸發指令-KPM6
      AND$=   D10600 "STC"  ; SECS_上位下指令暫存
      MOVP    D10540 D8610  ; 四色藍燈狀態
      OUT     M6200
488   LD      SM400  ; 常時 ON
      MPS
      AND=    D8610 K49
      OUT     M6510
      MRD
      AND=    D8610 K50
      OUT     M6511
      MPP
      AND=    D8610 K51
      OUT     M6512
504   LD      M6511
      LD      M6512
      AND     SM412  ; 1秒時鐘
      ORB
      ANI     M6510
      OUT     Y28  ; 四色燈  藍燈
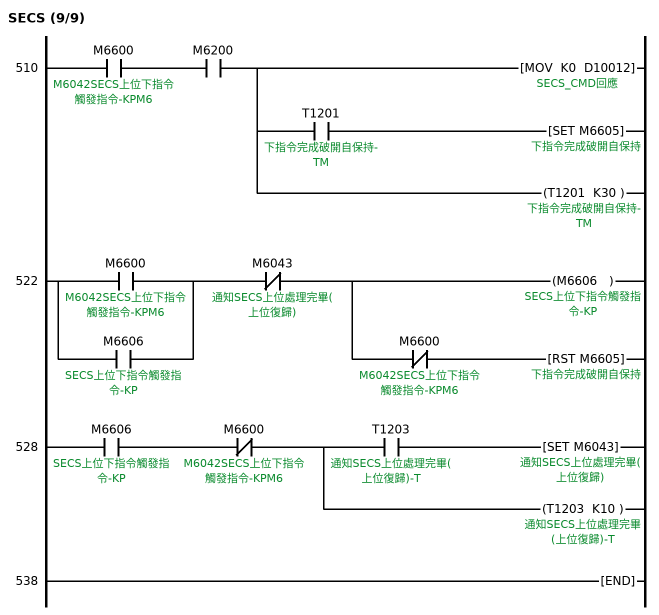
510   LD      M6600  ; M6042SECS上位下指令觸發指令-KPM6
      AND     M6200
      MOV     K0 D10012
      MPS
      AND     T1201  ; 下指令完成破開自保持-TM
      SET     M6605  ; 下指令完成破開自保持
      MPP
      OUT     T1201 K30  ; 下指令完成破開自保持-TM
522   LD      M6600  ; M6042SECS上位下指令觸發指令-KPM6
      OR      M6606  ; SECS上位下指令觸發指令-KP
      ANI     M6043  ; 通知SECS上位處理完畢(上位復歸)
      OUT     M6606  ; SECS上位下指令觸發指令-KP
      ANI     M6600  ; M6042SECS上位下指令觸發指令-KPM6
      RST     M6605  ; 下指令完成破開自保持
528   LD      M6606  ; SECS上位下指令觸發指令-KP
      ANI     M6600  ; M6042SECS上位下指令觸發指令-KPM6
      MPS
      AND     T1203  ; 通知SECS上位處理完畢(上位復歸)-T
      SET     M6043  ; 通知SECS上位處理完畢(上位復歸)
      MPP
      OUT     T1203 K10  ; 通知SECS上位處理完畢(上位復歸)-T
538   END
END_PROGRAM

// device comments not shown above
Y52  ; CH2輸出 允許/禁止標誌
Y53  ; CH3輸出 允許/禁止標誌
Y54  ; CH4輸出 允許/禁止標誌
Y55  ; CH5輸出 允許/禁止標誌
Y56  ; CH6輸出 允許/禁止標誌
Y57  ; CH7輸出 允許/禁止標誌
Y58  ; CH8輸出 允許/禁止標誌
M204  ; 批數歸零旗標
M270  ; 程式選擇#1
M271  ; 程式選擇#2
M272  ; 程式選擇#3
M273  ; 程式選擇#4
M274  ; 程式選擇#5
M275  ; 程式選擇#6
M276  ; 程式選擇#7
M277  ; 程式選擇#8
M278  ; 程式選擇#9
M279  ; 程式選擇#10
M280  ; 程式選擇#11
M281  ; 程式選擇#12
M282  ; 程式選擇#13
M283  ; 程式選擇#14
M284  ; 程式選擇#15
M285  ; 程式選擇#16
M286  ; 程式選擇#17
M287  ; 程式選擇#18
M288  ; 程式選擇#19
M289  ; 程式選擇#20
M1010  ; S:迴圈資料
M1011  ; 迴圈資料
M2000  ; 上位下達切換配方訊號
M2001  ; 配方搜尋成功
M2002  ; 配方搜尋失敗
M2003  ; 配方切換程序完成
M2005  ; 配方搜尋KP
M2011  ; 配方切換程序  1
M2012  ; 配方切換程序  2
M2013  ; 配方切換程序  3
M2014  ; 配方切換程序  4
M2015  ; 配方切換程序  5
M2016  ; 配方切換程序  6
M2017  ; 配方切換程序  7
M2018  ; 配方切換程序  8
M2019  ; 配方切換程序  9
M2020  ; 配方切換程序  10
M2060  ; 輸送啟動S
M2061  ; 輸送停止S
M2062  ; 點燈啟動S
M2063  ; 點燈停止S
M2105  ; 上位下PP判斷OK旗標
M2500  ; 維修保養畫面
M2502  ; PP_SEL完成旗標自保持
M2504  ; 爐內無版
M2505  ; PPSET_完成旗標
M4903  ; 爐內無板
M4920  ; 入口計數自保持
M4943  ; 上位下GO_REMOTE
M4944  ; 上位下GO-LOCAL
M4945  ; 上位允許放板START保持
M4946  ; 未達start 條件
M4948  ; 爐內片數=0
M4949  ; 機台自動生產中
M4950  ; 機台停止中(手動)
M4951  ; 上位允許切換配方自保持
M4952  ; S:切換配方動作流程切???
M4953  ; S:切換配方動作流程切啟動
M4954  ; S:手動狀態保持
M5120  ; 回上位Panel#1入板訊號
M5125  ; 回上位Panel#1出板訊號
M5204  ; 上位START-啟動
M5205  ; 上位STOP-停止
M5206  ; 上位允許切換配方
M5207  ; 上位切換成GO-REMOTE
M5208  ; 上位切換成GO-LOCAL
M5209  ; 上位下暫停進板
M5210  ; 上位下恢復進板
M5214  ; SECS上位下指令觸發Cmd-燈號
M5323  ; 緊急停止開關
M5901  ; SECS_上位下"START"
M5902  ; SECS_上位下"STOP"
M5903  ; SECS_上位下"LOCAL"
M5904  ; SECS_上位下"REMOTE"
M5905  ; SECS_上位下"PP_SELECT"
M6014  ; 配方同步SET M6058
M6058  ; 配方目錄同步R5300
M6059  ; Host刪除配方
M6060  ; Host刪除配方完成
M6102  ; 回上位機台狀態改變
M6103  ; 回上位自動啟動
M6104  ; 回上位當前使用配方變更
M6105  ; 回上位新增配方
M6106  ; 回上位刪除配方
M6107  ; 回上位修改配方
M6108  ; 回上位配方切換成功
M6109  ; 回上位Panel生產開始訊號
M6110  ; 回上位Panel生產結束訊號
M6111  ; 回上位Lot生產開始訊號
M6112  ; 回上位Lot生產結束訊號
M6113  ; 回上位配方狀態變更開始(開始升溫)
M6114  ; 回上位配方狀態變更結束(溫度到達)
M6115  ; PP_SELECT升溫中被中斷
M6116  ; SECS狀態改變中
M6117  ; 設備生產訊號收集-自動生產條件到
M6131  ; 生產完成程式結束
M6132  ; 機台狀態改變
M6134  ; 三色燈狀態改變
M6135  ; 回上位緊急停止開關訊號
M6136  ; 三色燈狀態改變
M6137  ; 手動
M6140  ; 要求上位回讀工單板號右爐
M6141  ; 要求上位回讀工單右爐
M6142  ; 三色黃燈
M6218  ; 和上位連線中
M6233  ; 上位要配方內容
M6320  ; FX機台狀態改變
M6820  ; 比對GO-REMOTE字串不對
M6821  ; 名稱GO-LOCAL比對不對
M6822  ; 比對RESUME字串不對
M6823  ; 比對PPID字串不對
M6824  ; 比對PAUSE字串不對
M6825  ; 比對START字串不對
M6826  ; 比對STOP字串不對
M6827  ; 比對PP_SELECT字串不對
M6860  ; 機台不在可生產狀態
M6861  ; 下STOP 機台不再READY/EXECUTING
M6862  ; 下PP_SELECT 機台不在待機中(IDLE)
M6863  ; 設備沒再暫停狀態
M6864  ; 機台不再START 狀態
M6865  ; 機台狀態不對
M6866  ; 設備沒再LOCAL狀態
M6867  ; 設備沒再REMOTE狀態
M7000  ; SECS_USE清除進板訊號
M7001  ; SECS_USE進板訊號ON
M7002  ; FX機台狀態改變保持
M7003  ; 急停RY KP
M7004  ; D10540=1(ASC) 滅燈
M7005  ; D10540=2(ASC) 亮燈
M7006  ; D10540=3(ASC)閃爍
M7007  ; 藍燈狀態變更旗標
M7008  ; 四色藍燈狀態變化完成RST
M7009  ; 四色藍燈狀態變化
M7010  ; S:迴圈資料
M7011  ; 迴圈資料
M7015  ; 上位OFF BZ
M7016  ; 上位 KP BZ
M7017  ; BZ狀態變化
M7023  ; 切換配方完成開始升溫旗標
M7040  ; START KP
M7041  ; STOP KP
M7042  ; PP_SELECT KP
M7100  ; SECS_上位下指令不為空
M7101  ; SECS_上位下"START"
M7102  ; SECS_上位下"STOP"
M7103  ; SECS_上位下"LOCAL"
M7104  ; SECS_上位下"REMOTE"
M7105  ; SECS_上位下"PP_SELECT"
M7120  ; 比對GO-REMOTE字串不對
M7121  ; 名稱GO-LOCAL比對不對
M7122  ; 比對RESUME字串不對
M7123  ; 比對PPID字串不對
M7124  ; 比對PAUSE字串不對
M7125  ; 比對START字串不對
M7126  ; 比對STOP字串不對
M7127  ; 比對PP_SELECT字串不對
M7130  ; [EH-02] 判斷配方ID不為零-1
M7131  ; [EH-02] 判斷配方ID不為零-2
M7132  ; [EH-02] 判斷配方ID無效
M7133  ; 判斷配方ID不為零=ON
M7134  ; 判斷配方ID不為空白=ON
M7140  ; [HH-02] 配方名稱搜尋KP
M7141  ; [HH-02] 配方名稱搜尋比對OK
M7142  ; [HH-02] 配方搜尋比對NG
M7150  ; [PPID]  判斷配方ID不為零-1
M7151  ; [PPID]  判斷配判斷配方ID不為零-2
M7152  ; [PPID]  判斷配方ID有效
M7160  ; [PPID]  配方搜尋KP
M7161  ; [PPID]  配方搜尋比對OK
M7162  ; [PPID]  配方搜尋比對NG
M7163  ; [PPID]  配方搜尋比對NG(空白)
M7170  ; [PPID]  配方搜尋比對OK_配方可
M7203  ; 未知?測試用
M7204  ; 上位允許放板START
M7205  ; 上位停止放板並清出料號
M7206  ; 上位允許切換配方
M7207  ; 上位切換成GO-REMOTE
M7208  ; 上位切換成GO-LOCAL
M7209  ; 上位下暫停進板
M7210  ; 上位下恢復進板
M7218  ; 和上位連線中
T95  ; 配方搜尋TM
T96  ; 配方切換程序完成TM
T217  ; S:切換配方旗標
D511  ; Temp1
D512  ; Temp2
D513  ; Temp3
D601  ; 月 PLC W
D602  ; 日 PLC W
D603  ; 時 PLC W
D604  ; 分 PLC W
D611  ; 月 PLC R
D612  ; 日 PLC R
D613  ; 時 PLC R
D614  ; 分 PLC R
D632  ; 配方組數
D811  ; #1      UV 燈開關
D812  ; #2      UV 燈開關
D813  ; #3      UV 燈開關
D814  ; #4      UV 燈開關
D2000  ; 上位下達切換配方名稱
D2011  ; 比對Bit 1-16組
D2012  ; 比對Bit 17-20組
D4000  ; S:爐內片數
D4002  ; 剩餘批次數量
D4007  ; PPSET_次數
D4008  ; Recipe  No.設定 -1
D4011  ; 上位下達切換配方名稱
D5439  ; PP_SEL- QTY-十位(DEC)
D5441  ; PP_SEL- QTY-個位(EDC)
D5443  ; PP_SEL- QTY-千位(DEC)
D5445  ; PP_SEL- QTY-百位(DEC)
D5447  ; PP_SEL- QTY-十萬位(DEC)
D5449  ; PP_SEL- QTY-萬位(DEC)
D5459  ; 從左數第一位
D5463  ; 從左數第二位
D5467  ; 從左數第三位
D5471  ; 從左數第四位
D5475  ; 從左數第五位
D5479  ; 從左數第六位
D5499  ; QTY數量
D5501  ; BF溫度配方NO比對不同時MOV同步
D5502  ; S:爐內片數
D5511  ; 配方組別計算暫存
D5512  ; 配方組別計算-1(-1)
D5514  ; 配方組別計算
D5520  ; S:剩餘批次數量
D5599  ; 判斷空白位置K0~19 BF
D6000  ; 配方設定號碼BF
D6002  ; Recipe  No.     (選擇)BF
D6034  ; 現在使用配方選擇組
D6720  ; 配方組迴圈+1
D6721  ; 配方迴圈內容+100
D7000  ; 讀出-PLC時間  年20xx    (DEC)
D7001  ; 讀出-PLC時間  月(DEC)
D7002  ; 讀出-PLC時間  日(DEC)
D7003  ; 讀出-PLC時間  時(DEC)
D7004  ; 讀出-PLC時間  分(DEC)
D7005  ; 讀出-PLC時間  秒(DEC)
D7006  ; 讀出-PLC時間  星期(DEC)
D7007  ; 讀出-PLC時間  年xx      (DEC)
D7010  ; 讀出-PLC時間  年xx      (BCD)
D7011  ; 讀出-PLC時間  月(BCD)
D7012  ; 讀出-PLC時間  日(BCD)
D7013  ; 讀出-PLC時間  時(BCD)
D7014  ; 讀出-PLC時間  分(BCD)
D7015  ; 讀出-PLC時間  秒(BCD)
D7016  ; 讀出-PLC時間  星期(BCD)
D7020  ; 讀出-PLC時間    年/月   (BCD)
D7021  ; 讀出-PLC時間    日/時   (BCD)
D7022  ; 讀出-PLC時間    分/秒   (BCD)
D7023  ; 讀出-PLC時間    星期    (BCD)
D7040  ; [ED-01] EQP Name#02/01
D7041  ; [ED-01] EQP Name#04/03
D7042  ; [ED-01] EQP Name#06/05
D7043  ; [ED-01] EQP Name#08/07
D7044  ; [ED-01] EQP Name#10/09
D7045  ; [ED-01] EQP Name#12/11
D7046  ; [ED-01] EQP Name#14/13
D7047  ; [ED-01] EQP Name#16/15
D7048  ; 總電量讀取*10(整數)-1
D7049  ; 總電量讀取*10(整數)-2
D7050  ; [ED-02] 配方異動上報數量暫存
D7059  ; [ED-02] Previous Index
D7080  ; EAP>EQP Month   (BCD)
D7081  ; EAP>EQP Year    (BCD)
D7082  ; EAP>EQP Hour    (BCD)
D7083  ; EAP>EQP Day     (BCD)
D7084  ; EAP>EQP Sec     (BCD)
D7085  ; EAP>EQP Min     (BCD)
D7086  ; EAP>EQP Week    (BCD)
D7087  ; EAP>EQP_EMPTY   (BCD)
D7090  ; EAP>EQP Year    (BIN)
D7091  ; EAP>EQP Month   (BIN)
D7092  ; EAP>EQP Day     (BIN)
D7093  ; EAP>EQP Hour    (BIN)
D7094  ; EAP>EQP Min     (BIN)
D7095  ; EAP>EQP Sec     (BIN)
D7096  ; EAP>EQP Week    (BIN)
D7097  ; EAP>EQP_EMPTY   (BIN)
D7099  ; [HC-01] PreviousIndex
D7100  ; [HC-02] CIM Msg 顯示形式
D7101  ; [HC-02] CIM Msg 顯示秒數
D7102  ; [HC-02] Type:0  等待上報筆數
D7103  ; [HC-02] Type:1  等待上報筆數
D7104  ; [HC-02] Type:0  顯示秒數換算暫存
D7105  ; [HC-02] Type:0  顯示秒數換算暫存
D7109  ; [HC-02] PreviousIndex
D7150  ; [EH-03] 變更回應
D7424  ; 烘烤時間(秒)
D7426  ; 烘烤時間(分)
D7500  ; HMI-IPT Recipe  NO. Set
D7501  ; Recipe  NO. Set (-1)
D7502  ; Recipe  NO. Set (上次)
D7508  ; [ED-02] 配方異動型態
D7509  ; Parameter Error
D7510  ; HMI-WIN 配方編輯寫入視窗
D7511  ; HMI-WIN 配方ID重覆視窗
D7512  ; 配方組別計算暫存
D7513  ; 配方組別計算-1(-1)
D7514  ; 配方組別計算-2-(1)
D7515  ; 配方組別計算
D7520  ; HMI-IPT 配方號碼選擇
D7521  ; 配方號碼選擇(-1)
D7700  ; [HH-04] RecipeID#02/01
D7701  ; [HH-04] RecipeID#04/03
D7702  ; [HH-04] RecipeID#06/05
D7703  ; [HH-04] RecipeID#08/07
D7704  ; [HH-04] RecipeID#10/09
D7705  ; [HH-04] RecipeID#12/11
D7706  ; [HH-04] RecipeID#14/13
D7707  ; [HH-04] RecipeID#16/15
D7708  ; [HH-04] RecipeID#18/17
D7709  ; [HH-04] RecipeID#20/19
D7710  ; [HH-04] RecipeID#22/21
D7711  ; [HH-04] RecipeID#24/23
D7712  ; [HH-04] RecipeID#26/25
D7713  ; [HH-04] RecipeID#28/27
D7714  ; [HH-04] RecipeID#30/29
D7720  ; [HH-04] Up      Heat    SV
D7721  ; [HH-04] Down    Heat    SV
D7722  ; [HH-04] ConveyorSpeed   SV
D7800  ; [ED-02] Modify  Type
D7801  ; [ED-02] RecipeID#02/01
D7802  ; [ED-02] RecipeID#04/03
D7803  ; [ED-02] RecipeID#06/05
D7804  ; [ED-02] RecipeID#08/07
D7805  ; [ED-02] RecipeID#10/09
D7806  ; [ED-02] RecipeID#12/11
D7807  ; [ED-02] RecipeID#14/13
D7808  ; [ED-02] RecipeID#16/15
D7809  ; [ED-02] RecipeID#18/17
D7810  ; [ED-02] RecipeID#20/19
D7811  ; [ED-02] RecipeID#22/21
D7812  ; [ED-02] RecipeID#24/23
D7813  ; [ED-02] RecipeID#26/25
D7814  ; [ED-02] RecipeID#28/27
D7815  ; [ED-02] RecipeID#30/29
D7821  ; [ED-02] Heat    SV      #01
D7822  ; [ED-02] Heat    SV      #02
D7823  ; [ED-02] Heat    SV      #03
D7824  ; [ED-02] HEAT-SV #04
D7825  ; [ED-02] HEAT-SV #05
D7826  ; [ED-02] HEAT-SV #06
D7827  ; [ED-02] 烘烤步進次數
D7828  ; [ED-02] 烘烤步進時間
D7829  ; [ED-02] 板材尺寸寬度設定
D10625  ; SECS_上位下STOP指令
D10640  ; SECS_上位下RESUME指令
D10675  ; SECS_上位下PPID指令
D10676  ; SECS_上位下PPID指令
W4C5  ; Modify  Type
W4C6  ; Recipe ID #02/#01
W4C7  ; Recipe ID #04/#03
W4C8  ; Recipe ID #06/#05
W4C9  ; Recipe ID #08/#07
W4CA  ; Recipe ID #10/#09
W4CB  ; Recipe ID #12/#11
W4CC  ; Recipe ID #14/#13
W4CD  ; Recipe ID #16/#15
W4CE  ; Recipe ID #18/#17
W4CF  ; Recipe ID #20/#19
W4D0  ; Recipe ID #22/#21
W4D1  ; Recipe ID #24/#23
W4D2  ; Recipe ID #26/#25
W4D3  ; Recipe ID #28/#27
W4D4  ; Recipe ID #30/#29
W4DA  ; Up-Heat SV
W4DB  ; Down-Heat SV
W4DC  ; Conyeyor Speed
W1600  ; Msg     Action  暫存1
W1601  ; CIM     Message 暫存1
W1640  ; Msg     Action  暫存2
P50  ; 來源轉浮點
P51  ; CALL迴圈結束旗標
P200  ; 判斷空白
P201  ; 判斷位置歸零
P202  ; 比對配方名給SV內容
P210  ; 轉浮點數
ZR138  ; 上報機台名稱MDLN
ZR145  ; 上報軟體編號SoftRev
ZR4135  ; 回應查詢配方內容組數
ZR4136  ; 上位下尋找配方名BF給SV內容
ZR4137  ; 上位下尋找配方名BF
ZR4151  ; 上位下PPID>查詢配方內容速度
ZR5300  ; PPID(Name)
ZR5302  ; PPID(Name)
